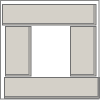
VISUALIZATION diaDataBox  // 100x100
    Button (4,77 96x21)
    Button (2,4 94x21)
    Button (5,26 26x50)
    Button (70,26 26x50)
END_VISUALIZATION

(* stored: Version 1.1.0.1, ProductVersion 3.1.4024.11
   Visu diaDataBox: Id {7408d88e-96f1-0460-201c-08e7c14b3b44} *)
